// TIA Portal V19 export
FUNCTION "M_CmpLT" : Bool   // FC15, LAD
TITLE = Module compare LOWER THAN / Module compare Lower than
// stored: Access Published, SetENOAutomatically false
   VAR_INPUT
      Xa : LReal;
      Xb : LReal;
      MODULE : LReal;
   END_VAR
BEGIN

REGION Network 1 (SCL): Xa < Xb return TRUE / Main
   #M_CmpLT := "M_PosAMinusPosB"(PosA := #Xa, PosB := #Xb, MODULE := #MODULE) < 0.0;
END_REGION
END_FUNCTION
